FUNCTION_BLOCK E_DELAY (* Delayed propagation of an event-Cancellable *)
  (* Standard: 61499-1; Classification: Event processing *)
  (* Version 0.1, 2001-04-05, JHC, Rockwell Automation, XML version *)
  (* Version 0.0, 1997-12-09, JHC, Rockwell Automation, SRC version *)
  (* Compiler header: package fb.rt.events; *)
  (* Compiler Java IBM VisualAge 3.0 *)
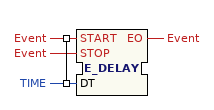
  EVENT_INPUT
    START WITH DT; (* Begin Delay *)
    STOP; (* Cancel Delay *)
  END_EVENT
  EVENT_OUTPUT
    EO; (* Delayed Event *)
  END_EVENT
  VAR_INPUT
    DT : TIME; (* Delay Time *)
  END_VAR
  SERVICE E_DELAY/RESOURCE
    SEQUENCE event_delay
      E_DELAY.START(DT) -> E_DELAY.EO();
    END_SEQUENCE
    SEQUENCE delay_canceled
      E_DELAY.START(DT);
      E_DELAY.STOP();
    END_SEQUENCE
    SEQUENCE no_multiple_delay
      E_DELAY.START(DT);
      E_DELAY.START(DT);
      -> E_DELAY.EO();
    END_SEQUENCE
  END_SERVICE
END_FUNCTION_BLOCK
